# EPICS substitutions: CryoControlApp/Db/plc_status.substitutions
file 1plc_status.vdb
{
         pattern { PLC_NAME            , AREA     , LOCA, CMPNUM }
                 { PLC_CP$(CP)2_CR1$(C), CP$(CP)2 , CR1$(C)  ,   4    }
}
